// TIA Portal V16 export
// export: Created 2023-02-28T11:29:00.7147107Z, ExportSetting WithDefaults, DisplayName Totally Integrated Automation Portal, DisplayVersion V16, DisplayName TIA Portal Version Control Interface, DisplayVersion V16, DisplayName TIA Portal Openness, DisplayVersion V16, DisplayName SINAMICS Startdrive Advanced, DisplayVersion V16, DisplayName SINAMICS Startdrive G130, G150, S120, S150, SINAMICS MV, S210, DisplayVersion V16, DisplayName SINAMICS Startdrive G110M, G120, G120C, G120D, G120P, DisplayVersion V16, DisplayName STEP 7 Professional, DisplayVersion V16, DisplayName STEP 7 Safety, DisplayVersion V16, DisplayName WinCC Professional, DisplayVersion V16
VAR_GLOBAL   // PLC tag table "Tabla de variables estándar"
   System_Byte AT %MB16383 : Byte;
   FirstScan AT %M16383.0 : Bool;
   DiagStatusUpdate AT %M16383.1 : Bool;
   AlwaysTRUE AT %M16383.2 : Bool;
   AlwaysFALSE AT %M16383.3 : Bool;
   Rojo AT %Q0.0 : Bool;
   Verde AT %Q0.1 : Bool;
   Amarillo AT %Q0.2 : Bool;
   X0 AT %M0.0 : Bool;
   X1 AT %M0.1 : Bool;
   X2 AT %M0.2 : Bool;
   X3 AT %M0.3 : Bool;
   PulsadorMarcha AT %I0.0 : Bool;
   T1 AT %T1 : Timer;
   T2 AT %T2 : Timer;
   T3 AT %T3 : Timer;
END_VAR
